{region '#Template'}
	{attribute 'Version' := '1.2.1.0'}
	{attribute 'Tags' := '"LCID": "1031", "Text": "Universal, Control, Event class, Notification"'}
	{attribute 'Tags' := '"LCID": "1033", "Text": "Universal, Control, Event class, Notification"'}
	{attribute 'Using' := '"Type": "Template", "URI": "EC_AMEV"'}
	{attribute 'Description' := '"LCID": "1031", "Text": "Ereignisklasse"'}
	{attribute 'Description' := '"LCID": "1033", "Text": "Event class"'}
{endregion}
FUNCTION_BLOCK FB_BA_EvtCategory EXTENDS FB_BA_View
VAR_INPUT CONSTANT
		EC				: FB_BA_EC;  
END_VAR

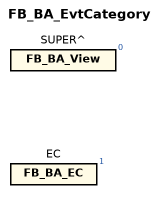
SUPER^(); // FB_BA_View
EC(); // FB_BA_EC

METHOD FB_init : BOOL
VAR_INPUT
	bInitRetains : BOOL; // if TRUE, the retain variables are initialized (warm start / cold start)
	bInCopyCode : BOOL;  // if TRUE, the instance afterwards gets moved into the copy code (online change)
END_VAR
EC.iParent					:= THIS^;
EC.iLabel					:= LblControl_EvtClass;	
EC.nInstanceID				:= EC_ID.NC10;
EC.sObjectName				:= '{Idx=10}';
EC.eEventType				:= E_BA_EventType.eAlarm;
EC.aPriority[1]				:= 16;
EC.aPriority[2]				:= 17;
EC.aPriority[3]				:= 18;
END_METHOD

END_FUNCTION_BLOCK

(* stored: Version 1.1.0.1, ProductVersion 3.1.4024.9
   POU FB_BA_EvtCategory: Id {9482cc0f-6ef0-4339-9176-e1ecba9fadd3}, SpecialFunc None
   Method FB_init: Id {58db39d5-cd29-47bd-a50e-dd077750d15e} *)
